Staubli VAL3: getPalletData.pgx

public program getPalletData(bool x_bCycle, TrajPallet& x_tTrajPallet)
begin
  // get the Pallet DATA
  if x_bCycle
    x_tTrajPallet=pt:tTraj[sTrajCycle]
  else
    x_tTrajPallet=pEditPoint
  endIf
end
